FUNCTION_BLOCK INFLUX_DB
  {SET_ATTRIBUTE(OpcUa, POINT.ENDPOINT)}
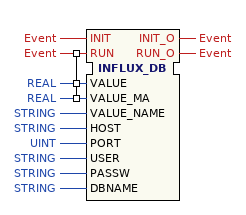
  EVENT_INPUT
    INIT;
    RUN WITH VALUE, VALUE_MA;
  END_EVENT
  EVENT_OUTPUT
    INIT_O;
    RUN_O;
  END_EVENT
  VAR_INPUT
    VALUE : REAL; {SET_ATTRIBUTE(OpcUa, Variable)}
    VALUE_MA : REAL; {SET_ATTRIBUTE(OpcUa, Variable)}
    VALUE_NAME : STRING; {SET_ATTRIBUTE(OpcUa, Constant)}
    HOST : STRING; {SET_ATTRIBUTE(OpcUa, Constant)}
    PORT : UINT; {SET_ATTRIBUTE(OpcUa, Constant)}
    USER : STRING; {SET_ATTRIBUTE(OpcUa, Constant)}
    PASSW : STRING; {SET_ATTRIBUTE(OpcUa, Constant)}
    DBNAME : STRING; {SET_ATTRIBUTE(OpcUa, Constant)}
  END_VAR
END_FUNCTION_BLOCK
